{attribute addProperty BoxType "KL2012"}
{attribute addProperty Id "OutputAT %Q*BOOL000"}
{attribute addProperty CRC "3881556014"}
{attribute addProperty SizeInBites "0"}
{attribute addProperty SizeInBytes "0"}
TYPE Channel_E75BD82E :
STRUCT
	{attribute addProperty Name "Output"}
	Output AT %Q* : BOOL;
END_STRUCT
END_TYPE

(* stored: Version 1.2.0.0, ProductVersion 3.1.4024.9
   DUT Channel_E75BD82E: Id {cffca111-49aa-4cc5-9eb2-902d781392ba} *)
